// TwinCAT 3 PLC project PlcProject
// ProgramVersion: 3.1.4026.16
// libraries:
//   Tc2_Standard, * (Beckhoff Automation GmbH)
//   Tc2_System, * (Beckhoff Automation GmbH)
// project tree:
//   GVLs/ GVL_CouplerOnDesk.TcGVL
//   / PlcTask.TcTTO
//   POUs/Hausaufgaben_SPH/ FB_AuFlankenauswertung.TcPOU, FB_AuFlipFlop.TcPOU
//   POUs/ MAIN.TcPOU
// real-time tasks:
//   TASK PlcTask: cycle T#10ms, priority 20, ADS port 350
// I/O:
//   DEVICE Master (EtherCAT), AmsNetId 192.168.10.102.2.1
//     Term 1 (EK1101) [EK1101 EtherCAT Coupler (2A E-Bus, ID switch)]
//       Digital Input (EL1014) [EL1014 4Ch. Dig. Input 24V, 10µs]
//       Digital Output (EL2004) [EL2004 4Ch. Dig. Output 24V, 0.5A]
//       Analog Input (EL3064) [EL3064 4Ch. Ana. Input 0-10V]
//       Analog Output (EL4102) [EL4102 2Ch. Ana. Output  0-10V, 16bit]
//       Display (EL6090) [EL6090 Displayklemme]
//       Endcover (EL9011)
// variable links:
//   (this object) <-> Master (EtherCAT)
//     PlcTask Inputs/GVL_CouplerOnDesk.bHotConnectGrpState <-> SyncUnits/[DeskGroup]/PlcTask/InfoData/State
//     PlcTask Inputs/GVL_CouplerOnDesk.bHotConnectGrpWcState <-> SyncUnits/[DeskGroup]/PlcTask/WcState/WcState
//     PlcTask Inputs/GVL_CouplerOnDesk.nEtherCatDevState <-> Inputs/DevState
//     PlcTask Inputs/GVL_CouplerOnDesk.nEtherCatSlaveCount <-> Inputs/SlaveCount
//   (this object) <-> Master (EtherCAT)/Term 1 (EK1101)
//     PlcTask Inputs/GVL_CouplerOnDesk.nCouplerId <-> ID/ID
//   (this object) <-> Master (EtherCAT)/Term 1 (EK1101)/Analog Input (EL3064)
//     PlcTask Inputs/GVL_CouplerOnDesk.nPotentiomerValue <-> AI Standard Channel 1/Value
//   (this object) <-> Master (EtherCAT)/Term 1 (EK1101)/Analog Output (EL4102)
//     PlcTask Outputs/GVL_CouplerOnDesk.nPotentiometerSupply <-> Channel 1/Output
//   (this object) <-> Master (EtherCAT)/Term 1 (EK1101)/Digital Input (EL1014)
//     PlcTask Inputs/GVL_CouplerOnDesk.bSelectorSwitch <-> Channel 1/Input
//     PlcTask Inputs/GVL_CouplerOnDesk.bSelectorSwitchLeftNC <-> Channel 2/Input
//     PlcTask Inputs/GVL_CouplerOnDesk.bSelectorSwitchRightNC <-> Channel 3/Input
//   (this object) <-> Master (EtherCAT)/Term 1 (EK1101)/Digital Output (EL2004)
//     PlcTask Outputs/GVL_CouplerOnDesk.bSelectorSwitchLed <-> Channel 1/Output
//   (this object) <-> Master (EtherCAT)/Term 1 (EK1101)/Display (EL6090)
//     PlcTask Inputs/GVL_CouplerOnDesk.bNavDown <-> DIS Inputs/Status/Down
//     PlcTask Inputs/GVL_CouplerOnDesk.bNavEnter <-> DIS Inputs/Status/Enter
//     PlcTask Inputs/GVL_CouplerOnDesk.bNavLeft <-> DIS Inputs/Status/Left
//     PlcTask Inputs/GVL_CouplerOnDesk.bNavRight <-> DIS Inputs/Status/Right
//     PlcTask Inputs/GVL_CouplerOnDesk.bNavUp <-> DIS Inputs/Status/Up
//     PlcTask Outputs/GVL_CouplerOnDesk.nDisplayRow1 <-> DIS Outputs/Value row 1
//     PlcTask Outputs/GVL_CouplerOnDesk.nDisplayRow2 <-> DIS Outputs/Value row 2

CONFIGURATION PlcProject
    RESOURCE PLC ON TwinCAT3
        TASK PlcTask(INTERVAL := T#10ms, PRIORITY := 20);
        PROGRAM MAIN WITH PlcTask : MAIN;
    END_RESOURCE
END_CONFIGURATION

// ---- GVLs/GVL_CouplerOnDesk.TcGVL
{attribute 'qualified_only'}
VAR_GLOBAL
    // Selector switch is activated (TRUE = left or right)
    bSelectorSwitch AT %I* : BOOL;
    // Selector switch is left (FALSE = left)
    bSelectorSwitchLeftNC AT %I* : BOOL;
    // Selector switch is right (FALSE = right)
    bSelectorSwitchRightNC AT %I* : BOOL;
    // Selector switch LED
    bSelectorSwitchLed AT %Q* : BOOL;
    // Potentiometer voltage tap
    nPotentiomerValue AT %I* : INT;
    // Potentiometer supply
    nPotentiometerSupply AT %Q* : INT;
    // Display navigation button Up
    bNavUp AT %I* : BOOL;
    // Display navigation button Down
    bNavDown AT %I* : BOOL;
    // Display navigation button Left
    bNavLeft AT %I* : BOOL;
    // Display navigation button Right
    bNavRight AT %I* : BOOL;
    // Display navigation button Enter
    bNavEnter AT %I* : BOOL;
    // Display row 1
    nDisplayRow1 AT %Q* : INT;
    // Display row 1
    nDisplayRow2 AT %Q* : INT;

    nEtherCatSlaveCount AT %I* : UINT;
    nEtherCatDevState AT %I* : UINT;
    bHotConnectGrpWcState AT %I* : BOOL;
    bHotConnectGrpState AT %I* : UINT;
    nCouplerId AT %I* : UINT;
END_VAR

// ---- POUs/MAIN.TcPOU
PROGRAM MAIN
VAR
    fbEdgeDetection : FB_AuFlankenauswertung;
END_VAR

fbEdgeDetection(Ix_Reset := NOT GVL_CouplerOnDesk.bSelectorSwitchLeftNC);

END_PROGRAM

// ---- POUs/Hausaufgaben_SPH/FB_AuFlankenauswertung.TcPOU
// Hausaufgabe, AU-011-002 Flankenauswertung
FUNCTION_BLOCK FB_AuFlankenauswertung
VAR_INPUT
    // Reset, TRUE = reset
    Ix_Reset : BOOL;
END_VAR
VAR_OUTPUT
    // Edge detected
    Mx_Imp_Reset : BOOL;
END_VAR
VAR
	// Status bit Reset input ist aktiv Variante 1
	bResetIsset: BOOL;
    // Instanz ansteigende Flankenauswertung Variante 2
    Mx_FP_Reset : R_TRIG;
    // Instanz fallende Flankenauswertung Variante 2
    Mx_FN_Reset : F_TRIG;
END_VAR

// Damit dieser Funktionsbaustein sinnvoll genutzt werden kann (beide Varianten führen die selbe Funktion aus, Ausgangsvariable
// bildet steigende und fallende Flanke ab), sollten nicht benötigte Programm-Varianten auskommentiert werden.
// Diese Code-Sammlung dient nur den Übungszwecken der Aufgabe "AU-011-002 Flankenauswertung".
// 
// Bezeichner welche nicht in der Aufgabenstellung vorgegeben sind entsprechen den folgenden Namenskonventionen:
//              https://infosys.beckhoff.com/content/1031/tc3_plc_intro/12073947403.html?id=915147275798565020
//

{region "Variante 1"}
// Setze Ausgang standardmässig zu FALSE
Mx_Imp_Reset := FALSE;

// Ansteigende Flankenerkennung
IF NOT bResetIsset AND Ix_Reset THEN
    Mx_Imp_Reset := TRUE;
END_IF

// Fallende Flankenerkennung
IF bResetIsset AND NOT Ix_Reset THEN
    Mx_Imp_Reset := TRUE;
END_IF

// Verknüpfung Reset Eingang mit Status bit
bResetIsset := Ix_Reset;
{endregion}

{region "Variante 2"}
// Ansteigende Flankenerkennung
Mx_FP_Reset(CLK := Ix_Reset);
// Fallende Flankenerkennung
Mx_FN_Reset(CLK := Ix_Reset);

// Zuweisung Ausgänge Ansteigende und Fallende Flankenerkennung
Mx_Imp_Reset := Mx_FP_Reset.Q OR Mx_FN_Reset.Q;
{endregion}

END_FUNCTION_BLOCK

// ---- POUs/Hausaufgaben_SPH/FB_AuFlipFlop.TcPOU
// Hausaufgabe, AU-011-001 FlipFlop
FUNCTION_BLOCK FB_AuFlipFlop
VAR_INPUT
    // Taster On, TRUE = On
    Ix_TasterOn : BOOL;
    // Taster Off, TRUE = Off
    Ix_TasterOff : BOOL;
END_VAR
VAR_OUTPUT
    // Ausgangsbit Anlage ein
    Mx_AnlageEin : BOOL;
END_VAR
VAR
    // Instanz Flip Flop Variante 2.1
    fbSetDominant : SR;
    // Instanz Flip Flop Variante 2.2
    fbResetDominant : RS;
END_VAR

// Damit dieser Funktionsbaustein sinnvoll genutzt werden kann (Ausgangsvariablen werden mehrmals
// beschrieben), müssen nicht benötigte Programm-Varianten auskommentiert werden.
// Diese Code-Sammlung dient nur den Übungszwecken der Aufgabe "AU-011-001 FlipFlop".
// 
// Bezeichner welche nicht in der Aufgabenstellung vorgegeben sind entsprechen den folgenden Namenskonventionen:
//              https://infosys.beckhoff.com/content/1031/tc3_plc_intro/12073947403.html?id=915147275798565020
//

// Variante 1.1, SET dominant
IF Ix_TasterOn THEN
    Mx_AnlageEin := TRUE;
ELSIF NOT Ix_TasterOff THEN
    Mx_AnlageEin := FALSE;
END_IF

// Variante 1.2, RESET dominant
IF Ix_TasterOff THEN
    Mx_AnlageEin := FALSE;
ELSIF Ix_TasterOn THEN
    Mx_AnlageEin := TRUE;
END_IF

// Variante 2.1, SET dominant
fbSetDominant(SET1 := Ix_TasterOn, RESET := NOT Ix_TasterOff);
Mx_AnlageEin := fbSetDominant.Q1;

// Variante 2.2, RESET dominant
fbResetDominant(SET := Ix_TasterOn, RESET1 := Ix_TasterOff);
Mx_AnlageEin := fbResetDominant.Q1;

END_FUNCTION_BLOCK
